// TwinCAT 3 PLC project Assignment_3_PLC
// ProgramVersion: 3.1.4024.0
// libraries:
//   Tc2_Standard, * (Beckhoff Automation GmbH)
//   Tc2_System, * (Beckhoff Automation GmbH)
//   Tc3_Module, * (Beckhoff Automation GmbH)
// project tree:
//   DUTs/ E_WashError.TcDUT, E_WashState.TcDUT, ST_MachineConfig.TcDUT
//   / PlcTask.TcTTO
//   POUs/ FB_HeavyWash.TcPOU, FB_NormalWash.TcPOU (not stored), FB_SoftWash.TcPOU (not stored), FB_WashingMachine.TcPOU (not stored), I_WashStrategy.TcIO, MAIN.TcPOU (not stored)
// real-time tasks:
//   TASK PlcTask: cycle T#10ms, priority 20, ADS port 350

CONFIGURATION Assignment_3_PLC
    RESOURCE PLC ON TwinCAT3
        TASK PlcTask(INTERVAL := T#10ms, PRIORITY := 20);
        PROGRAM MAIN WITH PlcTask : MAIN;
    END_RESOURCE
END_CONFIGURATION

// ---- DUTs/E_WashError.TcDUT
TYPE E_WashError :
(
    None,
    DoorOpenFault,
    WaterSupplyFault
);
END_TYPE

// ---- DUTs/E_WashState.TcDUT
TYPE E_WashState :
(
    Idle,
    Filling,
    Washing,
    Draining,
    Completed
);
END_TYPE

// ---- DUTs/ST_MachineConfig.TcDUT
TYPE ST_MachineConfig  :
STRUCT
	iDrumSpeed : INT;
	iWaterTemperature : INT;
END_STRUCT
END_TYPE

// ---- POUs/I_WashStrategy.TcIO
INTERFACE I_WashStrategy

METHOD GetDuration : TIME
END_METHOD

METHOD Start 
VAR_IN_OUT
    config : ST_MachineConfig;
END_VAR
END_METHOD

END_INTERFACE

// ---- POUs/FB_HeavyWash.TcPOU
FUNCTION_BLOCK FB_HeavyWash IMPLEMENTS I_WashStrategy

METHOD GetDuration : TIME
GetDuration := T#15S;
END_METHOD

METHOD Start 
VAR_IN_OUT
    config : ST_MachineConfig;
END_VAR
config.iDrumSpeed := 1200;
config.iWaterTemperature := 45;
END_METHOD

END_FUNCTION_BLOCK
